{attribute 'GeneratedUsingTerminal: EL6201-0000-0017'}
{attribute addProperty BoxType "EL6201-0000-0017"}
{attribute addProperty Id "Slave_28A_DI0BOOL1Slave_28A_DI1BOOL1Slave_28A_DI2BOOL1Slave_28A_DI3BOOL1Slave_28B_DI0BOOL1Slave_28B_DI1BOOL1Slave_28B_DI2BOOL1Slave_28B_DI3BOOL1"}
{attribute addProperty CRC "299083896"}
{attribute addProperty Size "8"}
TYPE Slave_28_Inputs_11D3A878 :
STRUCT
	{attribute addProperty Name "Slave_28A_DI0"}
	Slave_28A_DI0 : BOOL;
	{attribute addProperty Name "Slave_28A_DI1"}
	Slave_28A_DI1 : BOOL;
	{attribute addProperty Name "Slave_28A_DI2"}
	Slave_28A_DI2 : BOOL;
	{attribute addProperty Name "Slave_28A_DI3"}
	Slave_28A_DI3 : BOOL;
	{attribute addProperty Name "Slave_28B_DI0"}
	Slave_28B_DI0 : BOOL;
	{attribute addProperty Name "Slave_28B_DI1"}
	Slave_28B_DI1 : BOOL;
	{attribute addProperty Name "Slave_28B_DI2"}
	Slave_28B_DI2 : BOOL;
	{attribute addProperty Name "Slave_28B_DI3"}
	Slave_28B_DI3 : BOOL;
END_STRUCT
END_TYPE

(* stored: Version 1.2.0.0, ProductVersion 3.1.4024.9
   DUT Slave_28_Inputs_11D3A878: Id {f558fe0c-fc11-42f3-a344-04bff80f8d15} *)
